{attribute 'qualified_only'}
{attribute 'strict'}
{attribute  'hide'}
TYPE eWriteState :
(
	FileOpen_TRIGGER,
	FILE_OPEN,
	WAIT_FOR_EVENT,
	WRITE_EVENT_TRIGGER,
	WRITE_EVENT,
	FILE_CLOSE_TRIGGER,
	FILE_CLOSE,ERROR
);
END_TYPE

(* stored: Version 1.1.0.1, ProductVersion 3.1.4024.6
   EnumerationTextList eWriteState: Id {270a1658-b835-4b9a-90e0-4a09ad8d513c} *)
